// TIA Portal V18 export
VAR_GLOBAL   // PLC tag table "DI"
   in_SelStart AT %I0.0 : Bool;
   in_SelStop AT %I0.1 : Bool;
   in_BtnEmergency AT %I0.2 : Bool;
   in_BtnReset AT %I0.3 : Bool;
   in_Capacitive AT %I0.4 : Bool;
   in_5 AT %I0.5 : Bool;
   in_6 AT %I0.6 : Bool;
   in_PhCell_0 AT %I0.7 : Bool;
   in_PhCell_1 AT %I1.0 : Bool;
   in_PhCell_2 AT %I1.1 : Bool;
   in_PhCell_3 AT %I1.2 : Bool;
   in_PhCell_4 AT %I1.3 : Bool;
   in_PhCell_5 AT %I1.4 : Bool;
   in_PhCell_6 AT %I1.5 : Bool;
   in_PhCell_7 AT %I1.6 : Bool;
   in_PhCell_8 AT %I1.7 : Bool;
   in_Picker AT %I6.0 : Bool;
   in_17 AT %I6.1 : Bool;
   in_18 AT %I6.2 : Bool;
   in_19 AT %I6.3 : Bool;
   in_20 AT %I6.4 : Bool;
   in_21 AT %I6.5 : Bool;
   in_22 AT %I6.6 : Bool;
   in_23 AT %I6.7 : Bool;
   in_24 AT %I24.0 : Bool;
   in_25 AT %I24.1 : Bool;
   in_26 AT %I24.2 : Bool;
   in_27 AT %I24.3 : Bool;
   in_28 AT %I24.4 : Bool;
   in_29 AT %I24.5 : Bool;
   in_30 AT %I24.6 : Bool;
   in_31 AT %I24.7 : Bool;
END_VAR
